{attribute 'GeneratedUsingTerminal: EL3773-0000-0018'}
{attribute addProperty BoxType "EL3773-0000-0018"}
{attribute addProperty Id "I3_SamplesAT %I*I3_Samples_2D13B74B20"}
{attribute addProperty CRC "1788970028"}
{attribute addProperty Size "20"}
TYPE L3_Current_Samples_6AA1842C EXTENDS InputBase_8311D824 :
STRUCT
	{attribute addProperty Name "I3_Samples"}
	I3_Samples AT %I* : I3_Samples_2D13B74B;
END_STRUCT
END_TYPE

(* stored: Version 1.2.0.0, ProductVersion 3.1.4024.9
   DUT L3_Current_Samples_6AA1842C: Id {9a5216f4-3346-4def-b2f1-d67c2d6d8aee} *)
